TYPE TcoKukaRobotics_Config_v_5_x_x :
STRUCT
    InfoTime : TIME := T#2S;
    ErrorTime : TIME := T#0S;
END_STRUCT
END_TYPE

(* stored: Version 1.1.0.1, ProductVersion 3.1.4024.12
   DUT TcoKukaRobotics_Config_v_5_x_x: Id {eb448ab9-0eb5-0254-0c19-49c5799973df} *)
